# EPICS substitutions: caenDigitizerApp/Db/dt274x.substitutions
file "dt274x_base.db" { {} }

file "dt274x_ch.db" {
pattern { N }
{ "0" } { "1" }
}
